// SIMATIC S7-200 project (STEP 7-Micro/WIN), CPU 224 REL 01.11

SYMBOL_TABLE USER1
FORR             I0.0
REV              I0.1
STOPP            I0.2
THUAN            Q0.0
NGHICH           Q0.1
END_SYMBOL_TABLE

ORGANIZATION_BLOCK MAIN:OB1
TITLE=PROGRAM COMMENTS
BEGIN
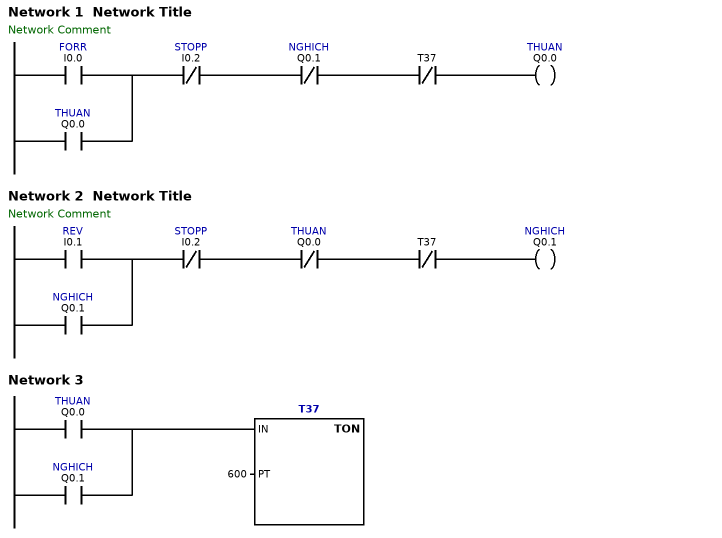
Network 1 // Network Title
// Network Comment
LD     FORR:I0.0
O      THUAN:Q0.0
AN     STOPP:I0.2
AN     NGHICH:Q0.1
AN     T37
=      THUAN:Q0.0
Network 2 // Network Title
// Network Comment
LD     REV:I0.1
O      NGHICH:Q0.1
AN     STOPP:I0.2
AN     THUAN:Q0.0
AN     T37
=      NGHICH:Q0.1
Network 3
LD     THUAN:Q0.0
O      NGHICH:Q0.1
TON    T37, 600
END_ORGANIZATION_BLOCK
